Staubli VAL3: cycle_searchPrg.pgx

program cycle_searchPrg(num x_nProg (dimensions=1), string& x_sProgName[] (dimensions=1), bool& x_bFound[] (dimensions=1))
  local num i
  local bool l_bOk
  local num l_nChar
  local num l_nProg
begin
  // init
  x_bFound=false
  x_sProgName=""
  //
  // get the list
  //
  // libList(saveData:sPathProg[0],sProgList)
  //
  // search the program from a number:
  //
  // "number+space+name"
  //
  // 01 MyPart
  // 10 YourPart
  //
  for i=0 to size(sProgList)-1
    if sProgList[i]!=""
      toNum(sProgList[i],l_nProg,l_bOk)
      if l_bOk and l_nProg==x_nProg
        x_sProgName=sProgList[i]
        x_bFound=true
        i=size(sProgList)-1
      endIf
    endIf
  endFor
end
